FUNCTION_BLOCK PUBLIC InputPortNotConnectedError EXTENDS Error
VAR
	state : (CLEARED, RAISED);
	port : I_InputPort;
END_VAR

PROPERTY Active : BOOL
GET
Active := state <> CLEARED;
END_GET
END_PROPERTY

METHOD PUBLIC Clear
port := 0;
state := CLEARED;
END_METHOD

PROPERTY PUBLIC ErrorCode : HRESULT
GET
ErrorCode := Tc2_System.E_HRESULTAdsErr.SYMBOLNOTFOUND;
END_GET
END_PROPERTY

PROPERTY Message : T_MaxString
GET
Message := 'Input port not connected';
END_GET
END_PROPERTY

METHOD PUBLIC Raise
VAR_INPUT
	Port : I_InputPort;
END_VAR
THIS^.port := Port;
state := RAISED;
END_METHOD

PROPERTY Reason : T_MaxString
GET
VAR
	message : STRING;
END_VAR
IF state = CLEARED THEN
	RETURN;
END_IF

Reason := port.Name;
END_GET
END_PROPERTY

END_FUNCTION_BLOCK

(* stored: Version 1.1.0.1, ProductVersion 3.1.4024.12
   POU InputPortNotConnectedError: Id {a9aca9eb-4d4e-0fe7-2725-b8601bc91b2d}, SpecialFunc None
   Property Active: Id {20dacd62-8743-05f0-3c18-e8d466902c6a}
   Get Get: Id {3cbcd73e-5293-02a1-0e43-ffd0b12811c6}
   Method Clear: Id {e4f6c949-0a3c-0b39-2976-4cfca73cc781}
   Property ErrorCode: Id {3e4f3eac-df0a-0738-3a38-5241491187a2}
   Get Get: Id {3eb1f540-7be6-0f27-0627-b2277b01249b}
   Property Message: Id {a79cdaa9-a00f-0bbb-1419-8ca11269f95c}
   Get Get: Id {b6073a34-82f2-07ab-07b4-1ed615d4082f}
   Method Raise: Id {607bc740-3a89-00d3-0198-7e2ea960ebdf}
   Property Reason: Id {ae2c560c-d56b-0f09-016d-71d5008526e2}
   Get Get: Id {aaa15406-0d20-0f38-1da9-6a652dd4b3ea} *)
